// TIA Portal project "WinCC_Learn" (V15.1)
// Este proyecto se crea para tomar pantallazos de los pasos de configuracion para la guia de PLC.

(* hardware
DEVICE "S7-1200 station_1"  S7-1200 Station
   slot 0: "Rack_0"  S7-1200 Rack  Rack  V1.0
   slot 1: "PLC_1"  CPU 1214C AC/DC/Rly  6ES7 214-1BG40-0XB0  V4.2
DEVICE "PC-System_1"  SIMATIC PC station
   slot 0: "Estación PC SIMATIC"  Rail  SIMATIC PC-Station  V1.0
      slot 125: "Stationmanager"  Station_Manager  V6.0.4
   slot 1: "HMI_RT_1"  WinCC RT Advanced  6AV2 104-0xxxx-xxxx  15.1.0.0
      slot 33792: "Interfaz host"  Host interface
   slot 2: "IE general_1"  IE General  IE_CP  V8.2.0
*)

// ===== PLC "PLC_1"  CPU 1214C AC/DC/Rly =====

VAR_GLOBAL   // PLC tag table "Tabla de variables estándar"
   "ArranqueMotorFisico" AT %I0.0 : Bool;
   "ParadaMotorFisico" AT %I0.1 : Bool;
   "ArranqueMotorVirtual" AT %M0.0 : Bool;
   "ParadaMotorVirtual" AT %M0.1 : Bool;
   "SalidaMotor" AT %Q0.0 : Bool;
END_VAR

ORGANIZATION_BLOCK "Main"   // OB1, LAD, ProgramCycle
TITLE = "Main Program Sweep (Cycle)"
{ S7_Optimized_Access := 'TRUE' }
VERSION : 0.1
   VAR_INPUT
      Initial_Call : Bool;   // Initial call of this OB
      Remanence : Bool;   // =True, if remanent data are available
   END_VAR
BEGIN

REGION Network 1
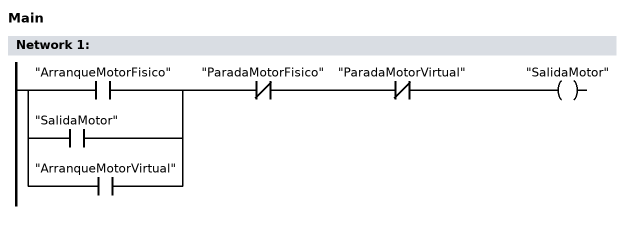
   RUNG wire#powerrail
      Contact( "ArranqueMotorFisico" )
      wire#w1
      I_Contact( "ParadaMotorFisico" )
      I_Contact( "ParadaMotorVirtual" )
      Coil( "SalidaMotor" )
   END_RUNG
   RUNG wire#powerrail
      Contact( "SalidaMotor" )
   END_RUNG wire#w1
   RUNG wire#powerrail
      Contact( "ArranqueMotorVirtual" )
   END_RUNG wire#w1
   // the same network as SCL:
   "SalidaMotor" := ("ArranqueMotorFisico" OR "SalidaMotor" OR "ArranqueMotorVirtual") AND NOT "ParadaMotorFisico" AND NOT "ParadaMotorVirtual";
END_REGION
END_ORGANIZATION_BLOCK

(* ===== HMI "HMI_RT_1" =====
system functions are stored by id; their names below are inferred from use
connection "HMI_Conexión_1": ETHERNET, S7_1200_OMS

HMI tags "Tabla de variables estándar"
   "ArranqueMotorVirtual" : Bool = PLC ArranqueMotorVirtual AT %M0.0, 1 s
   "ParadaMotorVirtual" : Bool = PLC ParadaMotorVirtual AT %M0.1, 1 s

screen "Imagen_1" 1024x768
   Button "Botón_1" at 107,152 size 165x59; TextOff 'M0.0'
      on Press: SetBit("ArranqueMotorVirtual")
   Button "Botón_2" at 337,153 size 165x59; TextOff 'M0.1'
      on Press: SetBit("ParadaMotorVirtual")
*)